// TIA Portal V18 export
// export: Created 2026-01-09T11:32:04.5013983Z, ExportSetting WithDefaults, DisplayName Totally Integrated Automation Portal, DisplayVersion V18 Update 5, DisplayName TIA Portal Openness, DisplayVersion V18 Update 5, DisplayName TIA Portal Teamcenter Gateway, DisplayVersion V18, DisplayName TIA Portal Version Control Interface, DisplayVersion V18, DisplayName SINAMICS Startdrive Advanced, DisplayVersion V18 SP2 Update 1, DisplayName SINAMICS Startdrive G110M, G120, G120C, G120D, G120P, G115D, DisplayVersion V18 SP2 Update 1, DisplayName SINAMICS Startdrive G130, G150, S120, S150, SINAMICS MV, S210, G220, S200, DisplayVersion V18 SP2 Update 1, DisplayName STEP 7 Professional, DisplayVersion V18 Update 5, DisplayName STEP 7 Safety, DisplayVersion V18, DisplayName WinCC Professional, DisplayVersion V18 Update 5
TagTable "PM_Count"
  PM_CountNG[0] : DInt  (%DB[PM_CountCycleDBNum].DBD["PM_CoNGAddress[0]"], CPU S71500-2PN_TP700, 1 s)
  PM_CountOK[2] : DInt  (%DB[PM_CountCycleDBNum].DBD["PM_CoOKAddress[2]"], CPU S71500-2PN_TP700, 1 s)
  PM_CountNG[2] : DInt  (%DB[PM_CountCycleDBNum].DBD["PM_CoNGAddress[2]"], CPU S71500-2PN_TP700, 1 s)
  PM_CountNG[7] : DInt  (%DB[PM_CountCycleDBNum].DBD["PM_CoNGAddress[7]"], CPU S71500-2PN_TP700, 1 s)
  PM_CountClearNG : Bool  (%DB[PM_CountCycleDBNum].DBX[PM_CoClearAddress].1, CPU S71500-2PN_TP700, 1 s)
  PM_CountTotal : DInt  (%DB[PM_CountCycleDBNum].DBD[PM_CoTotalAddress], CPU S71500-2PN_TP700, 1 s)
  PM_CountOK[1] : DInt  (%DB[PM_CountCycleDBNum].DBD["PM_CoOKAddress[1]"], CPU S71500-2PN_TP700, 1 s)
  PM_CountNG[4] : DInt  (%DB[PM_CountCycleDBNum].DBD["PM_CoNGAddress[4]"], CPU S71500-2PN_TP700, 1 s)
  PM_CountNG[1] : DInt  (%DB[PM_CountCycleDBNum].DBD["PM_CoNGAddress[1]"], CPU S71500-2PN_TP700, 1 s)
  PM_CountNG[3] : DInt  (%DB[PM_CountCycleDBNum].DBD["PM_CoNGAddress[3]"], CPU S71500-2PN_TP700, 1 s)
  PM_CountNG[6] : DInt  (%DB[PM_CountCycleDBNum].DBD["PM_CoNGAddress[6]"], CPU S71500-2PN_TP700, 1 s)
  PM_CountClearTotal : Bool  (%DB[PM_CountCycleDBNum].DBX[PM_CoClearAddress].2, CPU S71500-2PN_TP700, 1 s)
  PM_CountNG[5] : DInt  (%DB[PM_CountCycleDBNum].DBD["PM_CoNGAddress[5]"], CPU S71500-2PN_TP700, 1 s)
  PM_CountOK[0] : DInt  (%DB[PM_CountCycleDBNum].DBD["PM_CoOKAddress[0]"], CPU S71500-2PN_TP700, 1 s)
  PM_CountNG[8] : DInt  (%DB[PM_CountCycleDBNum].DBD["PM_CoNGAddress[8]"], CPU S71500-2PN_TP700, 1 s)
  PM_CountClearOK : Bool  (%DB[PM_CountCycleDBNum].DBX[PM_CoClearAddress].0, CPU S71500-2PN_TP700, 1 s)
  PM_CountCycleDBNum : UInt  (1 s)
  PM_CoClearAddress : UInt  (1 s)
  PM_CoNGAddress[1] : UInt  (1 s)
  PM_CoNGAddress[2] : UInt  (1 s)
  PM_CoNGAddress[3] : UInt  (1 s)
  PM_CoNGAddress[4] : UInt  (1 s)
  PM_CoNGAddress[0] : UInt  (1 s)
  PM_CoNGAddress[5] : UInt  (1 s)
  PM_CoNGAddress[6] : UInt  (1 s)
  PM_CoNGAddress[7] : UInt  (1 s)
  PM_CoNGAddress[8] : UInt  (1 s)
  PM_CoOKAddress[0] : UInt  (1 s)
  PM_CoOKAddress[1] : UInt  (1 s)
  PM_CoOKAddress[2] : UInt  (1 s)
  PM_CoTotalAddress : UInt  (1 s)
  PM_Num : USInt  (%DB[PM_CountCycleDBNum].DBB[PM_NumAddress], CPU S71500-2PN_TP700, 1 s)
  PM_NumAddress : UInt  (1 s)
